FUNCTION "ST10Cyl_interface61-70" : Void
VAR_INPUT
  AlwaysON : Bool;
  E_stop : Bool;
END_VAR
VAR_TEMP
  tTest : Bool;
END_VAR
BEGIN
  // Původní jazyk: LAD
  // Zdroj XML: EXPORT/Program blocks/OP010/10_Device/01_Cylinder/ST10Cyl_interface61-70.xml
  // (Žádný StructuredText network nebyl nalezen; LAD/STL/GRAPH není automaticky překládán.)
END_FUNCTION
